(* IEC 61131-3 sources: ATCMcontrol_Engineering/src/TargetBase/Libs/MECT, 7 files *)

(* ---- MECT_get_enquiry.st ---- *)
(*[[
    Alias="app_mect_enquiry",
    UserHelpURL= "ATCMfile:MECT_get_enquiry.HTML",
]]*)
FUNCTION MECT_get_enquiry : REAL (*[value read]*)
INLINE {STDLIB(MECT_get_enquiry)}
END_FUNCTION

(* ---- MECT_get_flag.st ---- *)
(*[[
    Alias="app_mect_flag",
    UserHelpURL= "ATCMfile:MECT_get_flag.HTML",
]]*)
FUNCTION MECT_get_flag : BYTE (*[flag]*)
INLINE {STDLIB(MECT_get_flag)}
END_FUNCTION

(* ---- MECT_get_status.st ---- *)
(*[[
    Alias="app_mect_status",
    UserHelpURL= "ATCMfile:MECT_get_status.HTML",
]]*)
FUNCTION MECT_get_status : INT (*[status]*)
INLINE {STDLIB(MECT_get_status)}
END_FUNCTION

(* ---- MECT_H_sread.st ---- *)
(*[[
    Alias="app_mect_enq",
    UserHelpURL= "ATCMfile:MECT_H_sread.HTML",
]]*)
FUNCTION MECT_H_sread : INT
VAR_INPUT
	id      : INT;                   (*[identifyer]*)
	command : STRING[2];             (*[command]*)
	width   : DINT;                  (*[protocol digit width]*)
END_VAR
INLINE {STDLIB(MECT_H_sread)}
END_FUNCTION

(* ---- MECT_H_swrite.st ---- *)
(*[[
    Alias="app_mect_hex_stx",
    UserHelpURL= "ATCMfile:MECT_H_swrite.HTML",
]]*)
FUNCTION MECT_H_swrite : INT
VAR_INPUT
	id      : INT;                   (*[identifyer]*)
	command : STRING[2];             (*[command]*)
	value   : INT;                   (*[value to write]*)
	width   : DINT;                  (*[protocol digit width]*)
END_VAR
INLINE {STDLIB(MECT_H_swrite)}
END_FUNCTION

(* ---- MECT_sread.st ---- *)
(*[[
    Alias="app_mect_enq",
    UserHelpURL= "ATCMfile:MECT_sread.HTML",
]]*)
FUNCTION MECT_sread : INT
VAR_INPUT
	id      : INT;                   (*[identifyer]*)
	command : STRING[2];             (*[command]*)
	width   : DINT;                  (*[protocol digit width]*)
END_VAR
INLINE {STDLIB(MECT_sread)}
END_FUNCTION

(* ---- MECT_swrite.st ---- *)
(*[[
    Alias="app_mect_float_stx",
    UserHelpURL= "ATCMfile:MECT_swrite.HTML",
]]*)
FUNCTION MECT_swrite : INT
VAR_INPUT
	id      : INT;                   (*[identifyer]*)
	command : STRING[2];             (*[command]*)
	value   : REAL;                  (*[value to write]*)
	width   : DINT;                  (*[protocol digit width]*)
END_VAR
INLINE {STDLIB(MECT_swrite)}
END_FUNCTION
